//{attribute 'qualified_only'}
VAR_GLOBAL
(* Pirani & Cold Cathode*)

    {attribute 'pytmc' :=' pv: MR2K4:KBO:GPI:01 '}
    {attribute 'TcLinkTo' := 	'.i_iPRESS_R	:=	TIIB[TMO_K4S2_DRL_02 (EK1100)]^K4S2_02_E1 (EL3174)^AI Standard Channel 2^Value '}
    MR2K4_KBO_GPI_01 : FB_MKS275;

    {attribute 'pytmc' :=' pv: MR2K4:KBO:GCC:01 '}
    {attribute 'TcLinkTo' := 	'.i_iPRESS_R	:=	TIIB[TMO_K4S2_DRL_02 (EK1100)]^K4S2_02_E1 (EL3174)^AI Standard Channel 3^Value;
                                 .i_xHV_ON	    :=	TIIB[TMO_K4S2_DRL_02 (EK1100)]^K4S2_02_E7 (EL1124)^Channel 3^Input;
                                 .i_xDisc_Active:=	TIIB[TMO_K4S2_DRL_02 (EK1100)]^K4S2_02_E7 (EL1124)^Channel 4^Input;
                                 .q_xHV_DIS		:= 	TIIB[TMO_K4S2_DRL_02 (EK1100)]^K4S2_02_E5 (EL2624)^Channel 2^Output	'}
    MR2K4_KBO_GCC_01 : FB_MKS500;

    {attribute 'pytmc' :=' pv: PA1K4:IP1:GPI:01 '}
    {attribute 'TcLinkTo' := 	'.i_iPRESS_R	:=	TIIB[TMO_K4S2_DRL_02 (EK1100)]^K4S2_02_E2 (EL3174)^AI Standard Channel 1^Value '}
    PA1K4_IP1_GPI_01 : FB_MKS275;


(*    {attribute 'pytmc' :=' pv: PA1K4:IP1:GCC:01 '}
    {attribute 'TcLinkTo' := 	'.i_iPRESS_R	:=	TIIB[TMO_K4S2_DRL_02 (EK1100)]^K4S2_02_E1 (EL3174)^AI Standard Channel 4^Value;
                                 .i_xHV_ON	    :=	TIIB[TMO_K4S2_DRL_02 (EK1100)]^K4S2_02_E8 (EL1124)^Channel 1^Input;
                                 .i_xDisc_Active:=	TIIB[TMO_K4S2_DRL_02 (EK1100)]^K4S2_02_E8 (EL1124)^Channel 2^Input;
                                 .q_xHV_DIS		:= 	TIIB[TMO_K4S2_DRL_02 (EK1100)]^K4S2_02_E5 (EL2624)^Channel 3^Output	'}
    PA1K4_IP1_GCC_01 : FB_MKS500;
*)
    {attribute 'pytmc' :=' pv: PA1K4:IP1:GCC:01 '}
    {attribute 'TcLinkTo' := 	'.i_iPRESS_R	:=	TIIB[TMO_K4S2_DRL_02 (EK1100)]^K4S2_02_E1 (EL3174)^AI Standard Channel 4^Value;
                                 .q_xHV_DIS		:= 	TIIB[TMO_K4S2_DRL_02 (EK1100)]^K4S2_02_E5 (EL2624)^Channel 3^Output	'}
    PA1K4_IP1_GCC_01 : FB_MX7M;
(*
    {attribute 'pytmc' :=' pv: IM4K4:PPM:GCC:01 '}
    {attribute 'TcLinkTo' := 	'.i_iPRESS_R	:=	TIIB[TMO_K4S2_DRL_02 (EK1100)]^K4S2_02_E2 (EL3174)^AI Standard Channel 2^Value;
                                 .i_xHV_ON	    :=	TIIB[TMO_K4S2_DRL_02 (EK1100)]^K4S2_02_E8 (EL1124)^Channel 3^Input;
                                 .i_xDisc_Active:=	TIIB[TMO_K4S2_DRL_02 (EK1100)]^K4S2_02_E8 (EL1124)^Channel 4^Input;
                                 .q_xHV_DIS		:= 	TIIB[TMO_K4S2_DRL_02 (EK1100)]^K4S2_02_E5 (EL2624)^Channel 4^Output	'}
    IM4K4_PPM_GCC_01 : FB_MKS500;
*)
    // replacing IM4K4_PPM_GCC_01 with CCM501
(*	{attribute 'pytmc' :=' pv: IM4K4:PPM:GCC:01 '}
    {attribute 'TcLinkTo' := 	'.i_iPRESS_R		:=	TIIB[TMO_K4S2_DRL_02 (EK1100)]^K4S2_02_E2 (EL3174)^AI Standard Channel 2^Value;
                                 .i_xHV_ON			:=	TIIB[TMO_K4S2_DRL_02 (EK1100)]^K4S2_02_E20A (EL1088)^Channel 1^Input;
                                 .q_xHV_DIS			:=	TIIB[TMO_K4S2_DRL_02 (EK1100)]^K4S2_02_E5 (EL2624)^Channel 4^Output '}
    IM4K4_PPM_GCC_01 : FB_CCM501;
*)
     {attribute 'pytmc' :=' pv: IM4K4:PPM:GCC:01 '}
    {attribute 'TcLinkTo' := 	'.i_iPRESS_R		:=	TIIB[TMO_K4S2_DRL_02 (EK1100)]^K4S2_02_E2 (EL3174)^AI Standard Channel 2^Value;
                                 .q_xHV_DIS			:=	TIIB[TMO_K4S2_DRL_02 (EK1100)]^K4S2_02_E5 (EL2624)^Channel 4^Output '}
    IM4K4_PPM_GCC_01 : FB_MX7M;


    {attribute 'pytmc' :=' pv: LI2K4:IP1:GFS:01 '}
    {attribute 'TcLinkTo' := 	'.i_iPRESS_R	:=	TIIB[B940_R20_EK0 (EK1100)]^R20_EK0_E1_MKS937B (EL3064)^AI Standard Channel 1^Value;
                                 .q_xHV_DIS		:=	TIIB[B940_R20_EK0 (EK1100)]^R20_EK0_E3_MKS937B (EL2794)^Channel 1^Output '}
    LI2K4_IP1_GFS_01 : FB_MKS422;

    {attribute 'pytmc' :=' pv: LI2K4:IP1:GFS:02 '}
    {attribute 'TcLinkTo' := 	'.i_iPRESS_R	:=	TIIB[B940_R20_EK0 (EK1100)]^R20_EK0_E1_MKS937B (EL3064)^AI Standard Channel 2^Value;
                                 .q_xHV_DIS		:=	TIIB[B940_R20_EK0 (EK1100)]^R20_EK0_E3_MKS937B (EL2794)^Channel 2^Output '}
    LI2K4_IP1_GFS_02 : FB_MKS422;

    {attribute 'pytmc' :=' pv: LI2K4:IP1:GFS:03 '}
    {attribute 'TcLinkTo' := 	'.i_iPRESS_R	:=	TIIB[B940_R20_EK0 (EK1100)]^R20_EK0_E2_MKS937B (EL3064)^AI Standard Channel 1^Value;
                                 .q_xHV_DIS		:=	TIIB[B940_R20_EK0 (EK1100)]^R20_EK0_E3_MKS937B (EL2794)^Channel 3^Output '}
    LI2K4_IP1_GFS_03 : FB_MKS422;


    {attribute 'pytmc' :=' pv: TM1K4:GCC:01 '}
    {attribute 'TcLinkTo' := 	'.i_iPRESS_R	:=	TIIB[TMO_K4S6_DRL_01 (EK1100)]^K4S6_01_E15 (EL3174)^AI Standard Channel 1^Value;
                                 .i_xHV_ON	    :=	TIIB[TMO_K4S6_DRL_01 (EK1100)]^K4S6_01_E20 (EL1124)^Channel 1^Input;
                                 .i_xDisc_Active:=	TIIB[TMO_K4S6_DRL_01 (EK1100)]^K4S6_01_E20 (EL1124)^Channel 2^Input;
                                 .q_xHV_DIS		:= 	TIIB[TMO_K4S6_DRL_01 (EK1100)]^K4S6_01_E14 (EL2624)^Channel 1^Output	'}
    TM1K4_GCC_01 : FB_MKS500;

 (*   {attribute 'pytmc' :=' pv: IM5K4:PPM:GCC:01 '}
    {attribute 'TcLinkTo' := 	'.i_iPRESS_R	:=	TIIB[TMO_K4S6_DRL_01 (EK1100)]^K4S6_01_E15 (EL3174)^AI Standard Channel 2^Value;
                                 .i_xHV_ON	    :=	TIIB[TMO_K4S6_DRL_01 (EK1100)]^K4S6_01_E20 (EL1124)^Channel 3^Input;
                                 .i_xDisc_Active:=	TIIB[TMO_K4S6_DRL_01 (EK1100)]^K4S6_01_E20 (EL1124)^Channel 4^Input;
                                 .q_xHV_DIS		:= 	TIIB[TMO_K4S6_DRL_01 (EK1100)]^K4S6_01_E14 (EL2624)^Channel 2^Output	'}
    IM5K4_PPM_GCC_01 : FB_MKS500;
*)
    {attribute 'pytmc' :=' pv: IM5K4:PPM:GCC:01 '}
    {attribute 'TcLinkTo' := 	'.i_iPRESS_R	:=	TIIB[TMO_K4S6_DRL_01 (EK1100)]^K4S6_01_E15 (EL3174)^AI Standard Channel 2^Value;
                                  .q_xHV_DIS		:= 	TIIB[TMO_K4S6_DRL_01 (EK1100)]^K4S6_01_E14 (EL2624)^Channel 2^Output	'}
    IM5K4_PPM_GCC_01 : FB_MX7M;

    // adding a new GPI here
    {attribute 'pytmc' :=' pv: IM5K4:PPM:GPI:01 '}
   {attribute 'TcLinkTo' := 	'.i_iPRESS_R	:=	TIIB[TMO_K4S6_DRL_01 (EK1100)]^K4S6_01_E18 (EL3174)^AI Standard Channel 3^Value '}
    IM5K4_IP1_GPI_01 : FB_MKS275;

    {attribute 'pytmc' :=' pv: PA2K4:IP1:GPI:01 '}
    {attribute 'TcLinkTo' := 	'.i_iPRESS_R	:=	TIIB[TMO_K4S6_DRL_01 (EK1100)]^K4S6_01_E15 (EL3174)^AI Standard Channel 4^Value '}
    PA2K4_IP1_GPI_01 : FB_MKS275;

    {attribute 'pytmc' :=' pv: PA2K4:IP1:GCC:01 '}
    {attribute 'TcLinkTo' := 	'.i_iPRESS_R	:=	TIIB[TMO_K4S6_DRL_01 (EK1100)]^K4S6_01_E15 (EL3174)^AI Standard Channel 3^Value;
                                 .i_xHV_ON	    :=	TIIB[TMO_K4S6_DRL_01 (EK1100)]^K4S6_01_E21 (EL1124)^Channel 1^Input;
                                 .i_xDisc_Active:=	TIIB[TMO_K4S6_DRL_01 (EK1100)]^K4S6_01_E21 (EL1124)^Channel 2^Input;
                                 .q_xHV_DIS		:= 	TIIB[TMO_K4S6_DRL_01 (EK1100)]^K4S6_01_E14 (EL2624)^Channel 3^Output	'}
    PA2K4_IP1_GCC_01 : FB_MKS500;


    {attribute 'pytmc' :=' pv: MR4K4:KBO:GPI:01 '}
    {attribute 'TcLinkTo' := 	'.i_iPRESS_R	:=	TIIB[TMO_K4S6_DRL_01 (EK1100)]^K4S6_01_E18 (EL3174)^AI Standard Channel 1^Value '}
    MR4K4_KBO_GPI_01 : FB_MKS275;

    {attribute 'pytmc' :=' pv: MR4K4:KBO:GCC:01 '}
    {attribute 'TcLinkTo' := 	'.i_iPRESS_R	:=	TIIB[TMO_K4S6_DRL_01 (EK1100)]^K4S6_01_E18 (EL3174)^AI Standard Channel 2^Value;
                                 .i_xHV_ON	    :=	TIIB[TMO_K4S6_DRL_01 (EK1100)]^K4S6_01_E21 (EL1124)^Channel 3^Input;
                                 .i_xDisc_Active:=	TIIB[TMO_K4S6_DRL_01 (EK1100)]^K4S6_01_E21 (EL1124)^Channel 4^Input;
                                 .q_xHV_DIS		:= 	TIIB[TMO_K4S6_DRL_01 (EK1100)]^K4S6_01_E14 (EL2624)^Channel 4^Output	'}
    MR4K4_KBO_GCC_01 : FB_MKS500;
    // need to update for the gauge model, if it is MKS500
    {attribute 'pytmc' :=' pv: TM2K4:KBO:GCC:01 '}
    {attribute 'TcLinkTo' := 	'.i_iPRESS_R	:=	TIIB[TMO_K4S8_DRL_02 (EK1100)]^K4S8_02_E4 (EL3174)^AI Standard Channel 1^Value;
                                 .i_xHV_ON	    :=	TIIB[TMO_K4S8_DRL_02 (EK1100)]^K4S8_02_E8 (EL1124)^Channel 1^Input;
                                 .i_xDisc_Active:=	TIIB[TMO_K4S8_DRL_02 (EK1100)]^K4S8_02_E8 (EL1124)^Channel 2^Input;
                                 .q_xHV_DIS		:= 	TIIB[TMO_K4S8_DRL_02 (EK1100)]^K4S8_02_E3 (EL2624)^Channel 1^Output'}
    TM2K4_KBO_GCC_01 : FB_MKS500;

    {attribute 'pytmc' :=' pv: TM2K4:KBO:GPI:01 '}
    {attribute 'TcLinkTo' := 	'.i_iPRESS_R	:=	TIIB[TMO_K4S8_DRL_02 (EK1100)]^K4S8_02_E4 (EL3174)^AI Standard Channel 3^Value '}
    TM2K4_KBO_GPI_01 : FB_MKS275;

(*
      // need to update for the gauge model, if it is MKS500
    {attribute 'pytmc' :=' pv: PF2K4:KBO:GCC:01 '}
    {attribute 'TcLinkTo' := 	'.i_iPRESS_R	:=	TIIB[TMO_K4S8_DRL_02 (EK1100)]^K4S8_02_E4 (EL3174)^AI Standard Channel 2^Value;
                                 .i_xHV_ON	    :=	TIIB[TMO_K4S8_DRL_02 (EK1100)]^K4S8_02_E8 (EL1124)^Channel 3^Input;
                                 .i_xDisc_Active:=	TIIB[TMO_K4S8_DRL_02 (EK1100)]^K4S8_02_E8 (EL1124)^Channel 4^Input;
                                 .q_xHV_DIS		:= 	TIIB[TMO_K4S8_DRL_02 (EK1100)]^K4S8_02_E3 (EL2624)^Channel 2^Output	'}
    PF2K4_WFS_GCC_01 : FB_MKS500;
*)
    // adding PF2K4_WFS_GCC_01 which is CCM501 type
(*    {attribute 'pytmc' :=' pv: PF2K4:KBO:GCC:01 '}
    {attribute 'TcLinkTo' := 	'.i_iPRESS_R		:=	TIIB[TMO_K4S8_DRL_02 (EK1100)]^K4S8_02_E4 (EL3174)^AI Standard Channel 2^Value;
                                 .i_xHV_ON			:=	TIIB[TMO_K4S8_DRL_02 (EK1100)]^K4S8_02_E6A (EL1084)^Channel 1^Input;
                                 .q_xHV_DIS			:=	TIIB[TMO_K4S8_DRL_02 (EK1100)]^K4S8_02_E3 (EL2624)^Channel 2^Output	'}
    PF2K4_WFS_GCC_01 : FB_CCM501;
*)
     {attribute 'pytmc' :=' pv: PF2K4:KBO:GCC:01 '}
    {attribute 'TcLinkTo' := 	'.i_iPRESS_R		:=	TIIB[TMO_K4S8_DRL_02 (EK1100)]^K4S8_02_E4 (EL3174)^AI Standard Channel 2^Value;
                                 .q_xHV_DIS			:=	TIIB[TMO_K4S8_DRL_02 (EK1100)]^K4S8_02_E3 (EL2624)^Channel 2^Output	'}
    PF2K4_WFS_GCC_01 : FB_MX7M;

(*
  // need to update for the gauge name and model
      {attribute 'pytmc' :=' pv: IM6K4:KBO:GPI:01 '}
    {attribute 'TcLinkTo' := 	'.i_iPRESS_R	:=	TIIB[TMO_K4S8_DRL_02 (EK1100)]^K4S8_02_E4 (EL3174)^AI Standard Channel 3^Value '}
    IM6K4_PPM_GPI_01 : FB_MKS275;
*)

(* Roughing gauges *)

    {attribute 'pytmc' :=' pv: TMO:ROUGH1:GPI:01 '}
    {attribute 'TcLinkTo' := 	'.i_iPRESS_R	:=	TIIB[TMO_WALL_WEST_EP01 (EP4374-0002)]^AI Inputs Channel 1^Value	'}
    TMO_ROUGH1_GPI_01 : FB_9XX;

    {attribute 'pytmc' :=' pv: TMO:ROUGH1:GPI:02 '}
    {attribute 'TcLinkTo' := 	'.i_iPRESS_R	:=	TIIB[TMO_K4S2_ EP1 (EP4374-0002)]^AI Inputs Channel 1^Value	'}
    TMO_ROUGH1_GPI_02 : FB_9XX;

    {attribute 'pytmc' :=' pv: TMO:ROUGH1:GPI:03 '}
    {attribute 'TcLinkTo' := 	'.i_iPRESS_R	:=	TIIB[TMO_K4S6_ EP1 (EP4374-0002)]^AI Inputs Channel 1^Value	'}
    TMO_ROUGH1_GPI_03 : FB_9XX;

    {attribute 'pytmc' :=' pv: TMO:ROUGH2:GPI:01 '}
    {attribute 'TcLinkTo' := 	'.i_iPRESS_R	:=	TIIB[TMO_WALL_WEST_EP01 (EP4374-0002)]^AI Inputs Channel 2^Value	'}
    TMO_ROUGH2_GPI_01 : FB_9XX;

    {attribute 'pytmc' :=' pv: TMO:ROUGH2:GPI:02 '}
    {attribute 'TcLinkTo' := 	'.i_iPRESS_R	:=	TIIB[TMO_K4S2_ EP1 (EP4374-0002)]^AI Inputs Channel 2^Value	'}
    TMO_ROUGH2_GPI_02 : FB_9XX;






END_VAR

(* stored: Version 1.1.0.1, ProductVersion 3.1.4024.12
   GVL GVL_Hutch_Gauges: Id {def8edf1-144c-4ec2-bb9e-c76eb49492a9} *)
